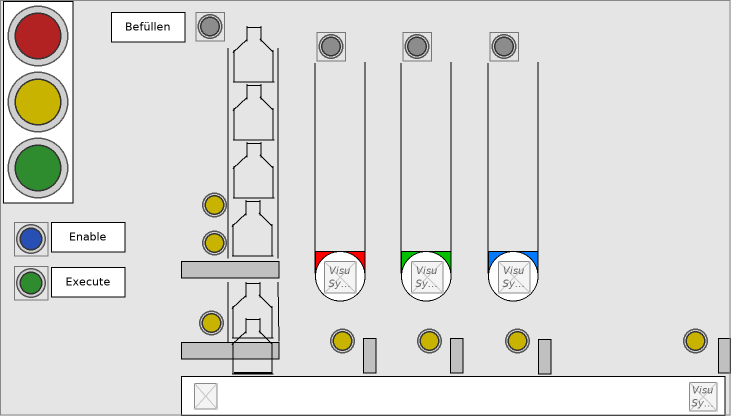
VISUALIZATION Visualization  // 731x416
    Rectangle (315,251 50x24)
        p2773130477: - MAIN.fbExt1.iFillLevel
    Lamp1 (200,190 29x30), variable: MAIN.bOut_VereinzelungNS1, style: Lamp-Lamp1-Yellow
    Lamp1 (200,228 29x30), variable: MAIN.bOut_VereinzelungNS2, style: Lamp-Lamp1-Yellow
    Lamp1 (197,308 29x30), variable: MAIN.bOut_VereinzelungNS3, style: Lamp-Lamp1-Yellow
    Group (3,1 70x202)
        Rectangle (0,0 70x202)
        Lamp1 (0,0 70x70), variable: MAIN.bIn_LedRot, style: Lamp-Lamp1-Red
        Lamp1 (0,66 70x70), variable: MAIN.bIn_LedYellow, style: Lamp-Lamp1-Yellow
        Lamp1 (0,132 70x70), variable: MAIN.bIn_LedGreen, style: Lamp-Lamp1-Green
    Line (228,258) (228,48)
    Line (278,258) (278,48)
    Line (279,341) (278,282)
    Line (228,342) (228,282)
    Rectangle (181,261 98x17)
        p3528305787: MAIN.fbVereinzelung.S1pos
        p874137650: MAIN.fbVereinzelung.S1pos
    Rectangle (181,342 98x17)
        p3528305787: MAIN.fbVereinzelung.S2pos
        p874137650: MAIN.fbVereinzelung.S2pos
    PushSwitch (12,222 38x34), variable: MAIN.bEnable, behaviour: TOGGLE, style: Switch-PushSwitch-Blue
    PushSwitch (12,266 38x34), variable: MAIN.bExecute, behaviour: TAP, style: Switch-PushSwitch-Green
    Rectangle (51,222 74x30), "Enable"
    Rectangle (51,267 74x30), "Execute"
    Group (232,200 41x57), invisible if: not MAIN.fbVereinzelung.fbSpeicherRohr.aSpeicher[0]
        Line (1,56) (1,24)
        Line (40,55) (40,24)
        Line (41,56) (0,56)
        Line (0,26) (14,13)
        Line (40,26) (27,13)
        Line (14,15) (14,0)
        Line (28,15) (28,0)
        Line (14,1) (28,1)
    Group (233,142 41x57), invisible if: Not MAIN.fbVereinzelung.fbSpeicherRohr.aSpeicher[1]
        Line (1,56) (1,24)
        Line (40,55) (40,24)
        Line (41,56) (0,56)
        Line (0,26) (14,13)
        Line (40,26) (27,13)
        Line (14,15) (14,0)
        Line (28,15) (28,0)
        Line (14,1) (28,1)
    Group (232,282 41x57), invisible if: not MAIN.bOut_VereinzelungNS3
        Line (1,56) (1,24)
        Line (40,55) (40,24)
        Line (41,56) (0,56)
        Line (0,26) (14,13)
        Line (40,26) (27,13)
        Line (14,15) (14,0)
        Line (28,15) (28,0)
        Line (14,1) (28,1)
    Group (233,84 41x57), invisible if: Not MAIN.fbVereinzelung.fbSpeicherRohr.aSpeicher[2]
        Line (1,56) (1,24)
        Line (40,55) (40,24)
        Line (41,56) (0,56)
        Line (0,26) (14,13)
        Line (40,26) (27,13)
        Line (14,15) (14,0)
        Line (28,15) (28,0)
        Line (14,1) (28,1)
    Group (233,26 41x57), invisible if: Not MAIN.fbVereinzelung.fbSpeicherRohr.aSpeicher[3]
        Line (1,56) (1,24)
        Line (40,55) (40,24)
        Line (41,56) (0,56)
        Line (0,26) (14,13)
        Line (40,26) (27,13)
        Line (14,15) (14,0)
        Line (28,15) (28,0)
        Line (14,1) (28,1)
    PushSwitch (194,12 32x29), variable: MAIN.fbVereinzelung.bBefullen, behaviour: TAP, style: Switch-PushSwitch-Gray
    RoundedRectangle (181,376 544x40)
    Lamp1 (328,326 29x30), variable: MAIN.bOUT_CnvNS1, style: Lamp-Lamp1-Yellow
    Lamp1 (503,326 29x30), variable: MAIN.bOUT_CnvNS3, style: Lamp-Lamp1-Yellow
    Lamp1 (415,326 29x30), variable: MAIN.bOUT_CnvNS2, style: Lamp-Lamp1-Yellow
    Lamp1 (681,326 29x30), variable: MAIN.bOUT_CnvNS4, style: Lamp-Lamp1-Yellow
    Group (232,318 41x57), invisible if: not MAIN.fbCNV.bBottleOnCNV
        p3560616238: MAIN.fbCNV.iBottlePos
        Line (1,56) (1,24)
        Line (40,55) (40,24)
        Line (41,56) (0,56)
        Line (0,26) (14,13)
        Line (40,26) (27,13)
        Line (14,15) (14,0)
        Line (28,15) (28,0)
        Line (14,1) (28,1)
    Rectangle (363,338 13x35), invisible if: MAIN.bIN_Stopper1
    Rectangle (450,338 13x35), invisible if: MAIN.bIN_Stopper2
    Rectangle (538,339 13x35), invisible if: MAIN.bIN_Stopper3
    Rectangle (718,338 13x35)
    Image (194,383 23x26), invisible if: not MAIN.fbCNV.bCNVisMoving, image: VisuSymbols.Symbols.ArrowHalfRightUp
    Image (689,382 28x29), invisible if: not MAIN.fbCNV.bCNVisMoving, image: VisuSymbols.Symbols.ArrowHalfRightDown
    Rectangle (111,12 74x30), "Befüllen"
    Ellipse (315,251 50x50)
    Line (315,273) (315,63)
    Line (365,272) (365,62)
    Rectangle (401,251 50x24)
        p2773130477: - MAIN.fbExt2.iFillLevel
    Ellipse (401,251 50x50)
    Line (401,273) (401,63)
    Line (451,272) (451,62)
    Rectangle (488,251 50x24)
        p2773130477: - MAIN.fbExt3.iFillLevel
    Ellipse (488,251 50x50)
    Line (488,273) (488,63)
    Line (538,272) (538,62)
    PushSwitch (315,32 32x29), variable: MAIN.bRefill1, behaviour: TAP, style: Switch-PushSwitch-Gray
    PushSwitch (401,32 32x29), variable: MAIN.bRefill2, behaviour: TAP, style: Switch-PushSwitch-Gray
    PushSwitch (488,32 32x29), variable: MAIN.bRefill3, behaviour: TAP, style: Switch-PushSwitch-Gray
    Image (324,261 32x32), invisible if: MAIN.fbExt1.NotMoving, image: VisuSymbols.Symbols.ArrowCircle2RightRightLeft
    Image (411,261 32x32), invisible if: MAIN.fbExt2.NotMoving, image: VisuSymbols.Symbols.ArrowCircle2RightRightLeft
    Image (498,261 32x32), invisible if: MAIN.fbExt3.NotMoving, image: VisuSymbols.Symbols.ArrowCircle2RightRightLeft
    Rectangle (234,372 38x1), invisible if: not MAIN.fbCNV.bBottleOnCNV
        p2773130477: - MAIN.fbBottleLevel.iFillLevel3 - MAIN.fbBottleLevel.iFillLevel1 - MAIN.fbBottleLevel.iFillLevel2
        p3560616238: MAIN.fbCNV.iBottlePos
        p1126004900: - MAIN.fbBottleLevel.iFillLevel1 - MAIN.fbBottleLevel.iFillLevel2
    Rectangle (234,372 38x1), invisible if: not MAIN.fbCNV.bBottleOnCNV
        p2773130477: - MAIN.fbBottleLevel.iFillLevel2 - MAIN.fbBottleLevel.iFillLevel1
        p3560616238: MAIN.fbCNV.iBottlePos
        p1126004900: - MAIN.fbBottleLevel.iFillLevel1
    Rectangle (234,372 38x1), invisible if: not MAIN.fbCNV.bBottleOnCNV
        p2773130477: - MAIN.fbBottleLevel.iFillLevel1
        p3560616238: MAIN.fbCNV.iBottlePos
END_VISUALIZATION

(* stored: Version 1.1.0.1
   Visu Visualization: Id {f4ba1731-bfd2-472e-a05a-c3f92ce7455e} *)
